// SIMATIC STEP 7 (V5.x) project TEMA 13 EJERCICIO 37
// CPU: CPU313 C-2 DP(1)
// station: P_ADR_BUS
// station: Hardware
// station: Equipo SIMATIC 300
// program: Programa S7(1)

SYMBOL_TABLE
"FLANCOS"	DB 1	DB 1
"MANIOBRA"	DB 2	DB 2
"SILO1 FC1 MIN."	I 0.0	BOOL
"SILO1 FC2 MAX."	I 0.1	BOOL
"SILO2 FC3 MIN."	I 0.2	BOOL
"SILO2 FC4 MAX."	I 0.3	BOOL
"Cycle Execution"	OB 1	OB 1
"TOLVA"	Q 0.0	BOOL
"TORNILLO SIN FIN"	Q 0.1	BOOL
"COMPUERTA SILO 1"	Q 0.2	BOOL
"CINTA SILO 1"	Q 0.3	BOOL
"COMPUERTA SILO 2"	Q 0.4	BOOL
"CINTA SILO 2"	Q 0.5	BOOL
END_SYMBOL_TABLE

DATA_BLOCK "FLANCOS"	// DB 1
VERSION : 0.1
  STRUCT
   M0 : BOOL ;
   M1 : BOOL ;
   M2 : BOOL ;
   M3 : BOOL ;
   M4 : BOOL ;
   M5 : BOOL ;
   M6 : BOOL ;
   M7 : BOOL ;
   M10 : BOOL ;
   M11 : BOOL ;
   M12 : BOOL ;
   M13 : BOOL ;
   M14 : BOOL ;
   M15 : BOOL ;
   M16 : BOOL ;
   M17 : BOOL ;
   M20 : BOOL ;
   M21 : BOOL ;
   M22 : BOOL ;
   M23 : BOOL ;
   M24 : BOOL ;
   M25 : BOOL ;
   M26 : BOOL ;
   M27 : BOOL ;
  END_STRUCT ;	
BEGIN
END_DATA_BLOCK

DATA_BLOCK "MANIOBRA"	// DB 2
VERSION : 0.1
  STRUCT
   M0 : BOOL ;
   M1 : BOOL ;
   M2 : BOOL ;
   M3 : BOOL ;
   M4 : BOOL ;
   M5 : BOOL ;
   M6 : BOOL ;
   M7 : BOOL ;
   M10 : BOOL ;
   M11 : BOOL ;
   M12 : BOOL ;
   M13 : BOOL ;
   M14 : BOOL ;
   M15 : BOOL ;
   M16 : BOOL ;
   M17 : BOOL ;
  END_STRUCT ;	
BEGIN
END_DATA_BLOCK

ORGANIZATION_BLOCK "Cycle Execution"	// OB 1
TITLE = "Main Program Sweep (Cycle)"
//ELEVACION Y CARGA DE SILOS DE GRANO
VERSION : 0.1
VAR_TEMP
  OB1_EV_CLASS : BYTE ;	//Bits 0-3 = 1 (Coming event), Bits 4-7 = 1 (Event class 1)
  OB1_SCAN_1 : BYTE ;	//1 (Cold restart scan 1 of OB 1), 3 (Scan 2-n of OB 1)
  OB1_PRIORITY : BYTE ;	//Priority of OB Execution
  OB1_OB_NUMBR : BYTE ;	//1 (Organization block 1, OB1)
  OB1_RESERVED_1 : BYTE ;	//Reserved for system
  OB1_RESERVED_2 : BYTE ;	//Reserved for system
  OB1_PREV_CYCLE : INT ;	//Cycle time of previous OB1 scan (milliseconds)
  OB1_MIN_CYCLE : INT ;	//Minimum cycle time of OB1 (milliseconds)
  OB1_MAX_CYCLE : INT ;	//Maximum cycle time of OB1 (milliseconds)
  OB1_DATE_TIME : DATE_AND_TIME ;	//Date and time OB1 started
END_VAR
BEGIN
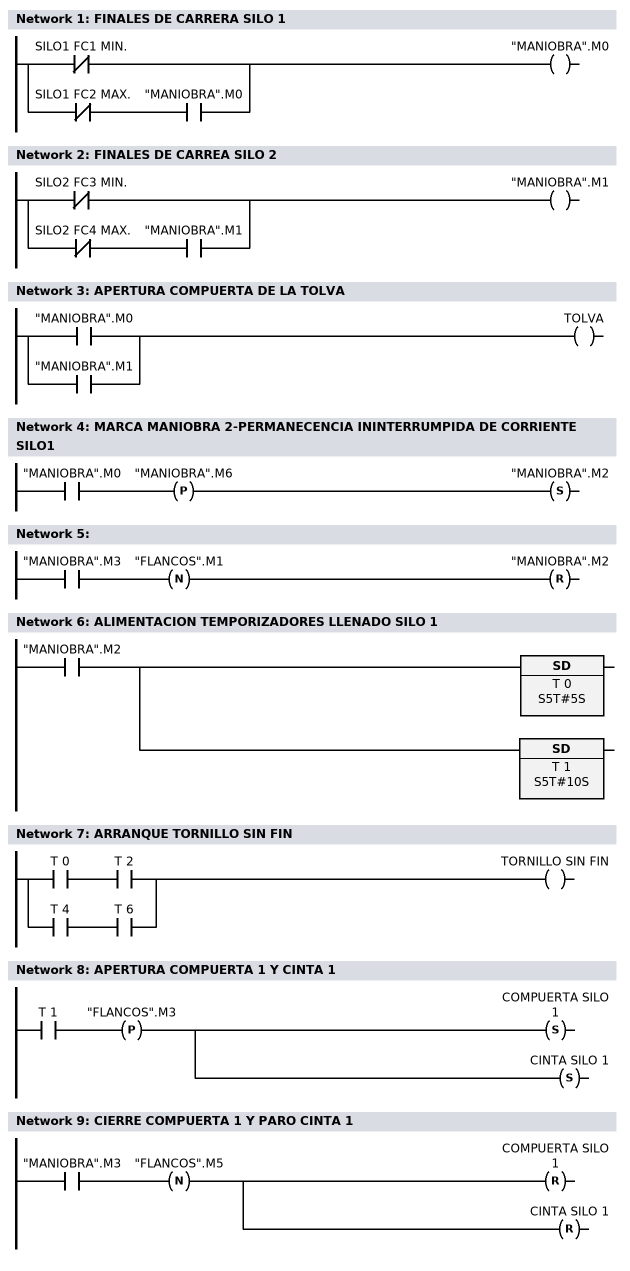
NETWORK
TITLE = FINALES DE CARRERA SILO 1 
//-FC1 MINIMO:SE ABRIRA CUANDO DETECTE GRANO Y SE CERRARA CUANDO NO LO DETECTE.
//-FC2 MAXIMO:"    "      "       "      "   "  "    "       "    "  "   "
//-MANIOBRA 0: SERA LA ENCARGADA DE ACTIVAR EL PROCESO DE ELEVACION Y CARGA 
//CUANDO 
//TENGA CORRIENTE.CUANDO NO LA TENGA INICIARA EL PROCESO DE DESCONEXION DE LOS 
//ELEMENTOS QUE INTERVENGAN EN EL PROCESO.
      ON    "SILO1 FC1 MIN.";
      O;
      AN    "SILO1 FC2 MAX.";
      A     "MANIOBRA".M0;
      =     "MANIOBRA".M0;
NETWORK
TITLE = FINALES DE CARREA SILO 2 
//-FC3 MINIMO:LA FUNCION ES LA MISMA QUE EN EL CASO ANTERIOR.
//-FC4 MAXIMO: "     "    "  "   "    "   "  "   "      "
//-MANIOBRA 1: "     "    "  "   "    "   "  "   "      "
//
      ON    "SILO2 FC3 MIN.";
      O;
      AN    "SILO2 FC4 MAX.";
      A     "MANIOBRA".M1;
      =     "MANIOBRA".M1;
NETWORK
TITLE = APERTURA COMPUERTA DE LA TOLVA
      O     "MANIOBRA".M0;
      O     "MANIOBRA".M1;
      =     "TOLVA";
NETWORK
TITLE = MARCA MANIOBRA 2-PERMANECENCIA ININTERRUMPIDA DE CORRIENTE SILO1
      A     "MANIOBRA".M0;
      FP    "MANIOBRA".M6;
      S     "MANIOBRA".M2;
NETWORK
TITLE =
      A     "MANIOBRA".M3;
      FN    "FLANCOS".M1;
      R     "MANIOBRA".M2;
NETWORK
TITLE = ALIMENTACION TEMPORIZADORES LLENADO SILO 1 
      A     "MANIOBRA".M2;
      L     S5T#5S;
      SD    T 0;
      L     S5T#10S;
      SD    T 1;
NETWORK
TITLE = ARRANQUE TORNILLO SIN FIN
      A     T 0;
      A     T 2;
      O;
      A     T 4;
      A     T 6;
      =     "TORNILLO SIN FIN";
NETWORK
TITLE = APERTURA COMPUERTA 1 Y CINTA 1 
      A     T 1;
      FP    "FLANCOS".M3;
      S     "COMPUERTA SILO 1";
      S     "CINTA SILO 1";
NETWORK
TITLE = CIERRE COMPUERTA 1 Y PARO CINTA 1
      A     "MANIOBRA".M3;
      FN    "FLANCOS".M5;
      R     "COMPUERTA SILO 1";
      R     "CINTA SILO 1";
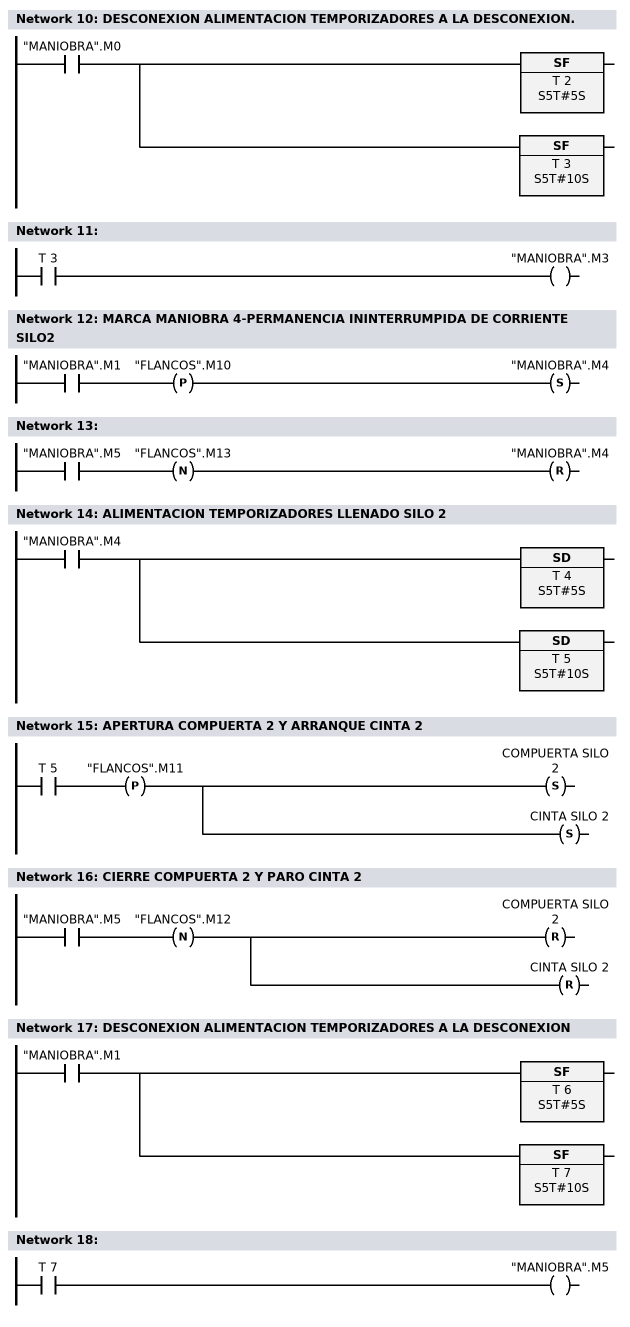
NETWORK
TITLE = DESCONEXION ALIMENTACION TEMPORIZADORES A LA DESCONEXION.
      A     "MANIOBRA".M0;
      L     S5T#5S;
      SF    T 2;
      L     S5T#10S;
      SF    T 3;
NETWORK
TITLE =
      A     T 3;
      =     "MANIOBRA".M3;
NETWORK
TITLE = MARCA MANIOBRA 4-PERMANENCIA ININTERRUMPIDA DE CORRIENTE SILO2
      A     "MANIOBRA".M1;
      FP    "FLANCOS".M10;
      S     "MANIOBRA".M4;
NETWORK
TITLE =
      A     "MANIOBRA".M5;
      FN    "FLANCOS".M13;
      R     "MANIOBRA".M4;
NETWORK
TITLE = ALIMENTACION TEMPORIZADORES LLENADO SILO 2
      A     "MANIOBRA".M4;
      L     S5T#5S;
      SD    T 4;
      L     S5T#10S;
      SD    T 5;
NETWORK
TITLE = APERTURA COMPUERTA 2 Y ARRANQUE CINTA 2 
      A     T 5;
      FP    "FLANCOS".M11;
      S     "COMPUERTA SILO 2";
      S     "CINTA SILO 2";
NETWORK
TITLE = CIERRE COMPUERTA 2 Y PARO CINTA 2 
      A     "MANIOBRA".M5;
      FN    "FLANCOS".M12;
      R     "COMPUERTA SILO 2";
      R     "CINTA SILO 2";
NETWORK
TITLE = DESCONEXION ALIMENTACION TEMPORIZADORES A LA DESCONEXION 
      A     "MANIOBRA".M1;
      L     S5T#5S;
      SF    T 6;
      L     S5T#10S;
      SF    T 7;
NETWORK
TITLE =
      A     T 7;
      =     "MANIOBRA".M5;
END_ORGANIZATION_BLOCK
